FUNCTION_BLOCK Module_Mockup EXTENDS Module
VAR
	_WasCalled : BOOL;
END_VAR

METHOD GetComponentByName : I_Component
VAR_INPUT
	Name : T_MaxString;
END_VAR
GetComponentByName := ComponentCollection.GetComponentByName(Name);
END_METHOD

METHOD GetModuleByName : I_Module
VAR_INPUT
	Module : T_MaxString;
END_VAR
GetModuleByName := ModuleCollection.GetModuleByName(Module);
END_METHOD

(* This Module will be done initializeing when ModuleInitialized := TRUE;, subequently all subitems will be called to be initialized*)
METHOD Initializing
ModuleInitialized := TRUE;
END_METHOD

METHOD OnCyclicCall
END_METHOD

PROPERTY WasCalled : BOOL
GET
WasCalled := _WasCalled;
END_GET
END_PROPERTY

END_FUNCTION_BLOCK

(* stored: Version 1.1.0.1, ProductVersion 3.1.4026.18
   POU Module_Mockup: Id {7a19c327-6901-4f31-9929-3e5451c7fded}, SpecialFunc None
   Method GetComponentByName: Id {990722a9-e6ba-42d8-a534-ad8a1a576b42}
   Method GetModuleByName: Id {05f0c2db-c3ab-4ec2-811c-8f7d2cab20c6}
   Method Initializing: Id {bc232e85-fa48-4c06-a04a-c2ed6effeb30}
   Method OnCyclicCall: Id {6289fb49-0027-4053-924c-aef8e019c7f1}
   Property WasCalled: Id {91085036-5c6f-4b58-9a52-0384d5935b37}
   Get Get: Id {ab795f9e-581c-453c-9d38-d018af0dfa2d} *)
